// Mitsubishi GX Works2 project: Analog   PLC: Q03UDV

PROGRAM MAIN
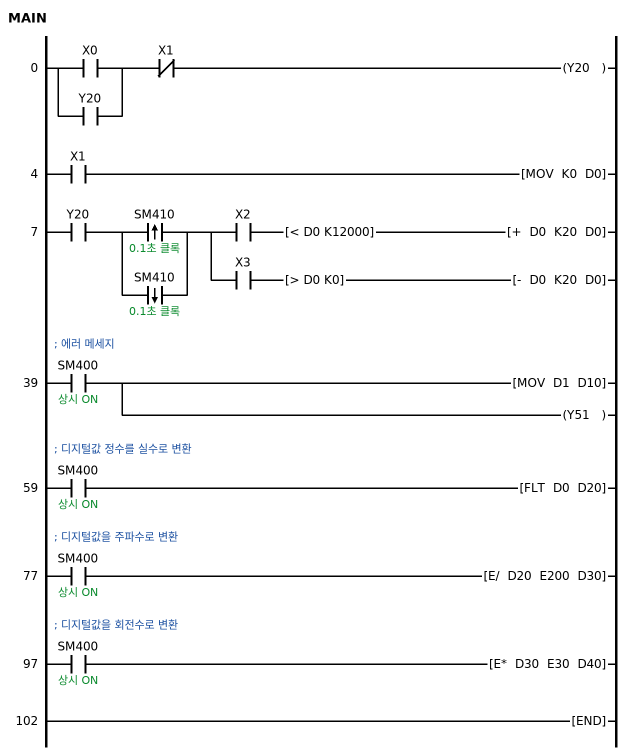
0     LD      X0
      OR      Y20
      ANI     X1
      OUT     Y20
4     LD      X1
      MOV     K0 D0
7     LD      Y20
      LDP     SM410  ; 0.1초 클록
      ORF     SM410  ; 0.1초 클록
      ANB
      MPS
      AND     X2
      AND<    D0 K12000
      +       D0 K20 D0
      MPP
      AND     X3
      AND>    D0 K0
      -       D0 K20 D0
; 에러 메세지
39    LD      SM400  ; 상시 ON
      MOV     D1 D10
      OUT     Y51
; 디지털값 정수를 실수로 변환
59    LD      SM400  ; 상시 ON
      FLT     D0 D20
; 디지털값을 주파수로 변환
77    LD      SM400  ; 상시 ON
      E/      D20 E200 D30
; 디지털값을 회전수로 변환
97    LD      SM400  ; 상시 ON
      E*      D30 E30 D40
102   END
END_PROGRAM
